{attribute 'GeneratedUsingTerminal: EK1122-0000-0018'}
{attribute addProperty BoxType "EK1122-0000-0018"}
{attribute addProperty Id "RC40_VI_AES_D_BC_ECAT_xAES_A3B0707168RC40_SAFETY_Flexi_Soft_EtherCAT_GatewayFlexi_Soft_EtherCAT_Gateway_DE394EDD5"}
{attribute addProperty CRC "3942309064"}
{attribute addProperty Size "73"}
{attribute addProperty Name "RC40_A2 (EK1122)"}
TYPE RC40_A2_EK1122_EAFADCC8 EXTENDS EK1122_1FC0878B :
STRUCT
	{attribute addProperty Name "RC40_VI (AES-D-BC-ECAT)"}
	{attribute addProperty PreviousPort "RC40_A2 (EK1122) : D"}
	{attribute addProperty SyncUnit "C40"}
	RC40_VI_AES_D_BC_ECAT_x : AES_A3B07071;
	{attribute addProperty Name "RC40_SAFETY (Flexi Soft EtherCAT Gateway)"}
	{attribute addProperty PreviousPort "RC40_A2 (EK1122) : B"}
	{attribute addProperty SyncUnit "C40"}
	RC40_SAFETY_Flexi_Soft_EtherCAT_Gateway : Flexi_Soft_EtherCAT_Gateway_DE394EDD;
END_STRUCT
END_TYPE

(* stored: Version 1.2.0.0, ProductVersion 3.1.4024.11
   DUT RC40_A2_EK1122_EAFADCC8: Id {22d0a313-d0b1-0fbc-3e2b-2ebcfc0ea0d6} *)
